{attribute 'linkalways'} 
{attribute 'no_explicit_call' := 'This FB is a CLASS and must be accessed using methods or properties'}
{attribute 'enable_dynamic_creation'}
FUNCTION_BLOCK Node_F_VN_ResetRoi EXTENDS VisionNode
VAR
    ipImage : _ITcVnImage;
    hrPrev : _HRESULT(S_OK);
	hresult : _HRESULT(S_OK);
END_VAR

METHOD PUBLIC  Clone : I_Node
VAR
	pNode : POINTER TO Node_F_VN_ResetRoi;
END_VAR
pNode := __NEW(Node_F_VN_ResetRoi);
Clone := pNode^;
END_METHOD

METHOD FB_init : BOOL
VAR_INPUT
	bInitRetains : BOOL; // if TRUE, the retain variables are initialized (warm start / cold start)
	bInCopyCode : BOOL;  // if TRUE, the instance afterwards gets moved into the copy code (online change)
END_VAR
AddInput('ipImage', ipImage);
AddOutput('ipImage', ipImage);
AddOutput('hresult',hresult);
END_METHOD

METHOD PROTECTED  OnExecute : HRESULT
hresult.Value := F_VN_ResetRoi(
    ipImage := ipImage.Value,
	hrPrev:= hrPrev.Value);
END_METHOD

METHOD PUBLIC PreExecutionCheck
VAR_INPUT
	Check : I_PreExecutionChecks;
END_VAR
IF FAILED(hrPrev.Value) THEN
    RETURN;
END_IF

Check.IsTrue(ipImage.IsValid, 'ipImage must contain an image');
END_METHOD

END_FUNCTION_BLOCK

(* stored: Version 1.1.0.1, ProductVersion 3.1.4024.13
   POU Node_F_VN_ResetRoi: Id {945b306f-8a1f-0f17-1a95-71bc89a62646}, SpecialFunc None
   Folder Constructor: Id {d38f6118-a90b-033d-2918-8e6f977b098b}
   Method Clone: Id {c0e41d5e-5a39-0a8a-22ee-dd5529cbf5c3}
   Method FB_init: Id {f1ecd4fe-3c43-0c64-15ac-19e2ffe5cc65}
   Method OnExecute: Id {0c1fd4a6-97f0-03c0-0235-3ff2feb131ab}
   Method PreExecutionCheck: Id {711b1086-8956-0fcc-3f40-65f7c9dbb587} *)
